FUNCTION_BLOCK EnableCheck (* Template for an empty basic function block *)
  (* Standard: 61499-2 *)
  (* Version 1.0, 2018-06-08, Duc Do Tran, OFFIS e.V. *)
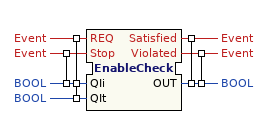
  EVENT_INPUT
    REQ WITH QIi, QIt;
    Stop WITH QIi;
  END_EVENT
  EVENT_OUTPUT
    Satisfied WITH OUT;
    Violated WITH OUT;
  END_EVENT
  VAR_INPUT
    QIi : BOOL := 1; (* QIt *)
    QIt : BOOL;
  END_VAR
  VAR_OUTPUT
    OUT : BOOL;
  END_VAR
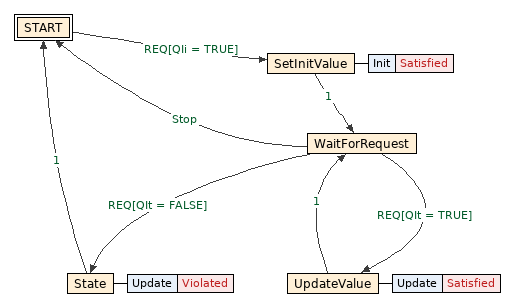
  EC_STATES
    START; (* Initial State *)
    SetInitValue : Init -> Satisfied;
    UpdateValue : Update -> Satisfied;
    WaitForRequest;
    State : Update -> Violated;
  END_STATES
  EC_TRANSITIONS
    START TO SetInitValue := REQ[QIi = TRUE];
    SetInitValue TO WaitForRequest := 1;
    WaitForRequest TO UpdateValue := REQ[QIt = TRUE];
    UpdateValue TO WaitForRequest := 1;
    WaitForRequest TO START := Stop;
    WaitForRequest TO State := REQ[QIt = FALSE];
    State TO START := 1;
  END_TRANSITIONS
  ALGORITHM Init IN ST: (* new algorithm *)
OUT := QIi;
  END_ALGORITHM
  ALGORITHM Update IN ST: (* new algorithm *)
OUT := QIt;
  END_ALGORITHM
END_FUNCTION_BLOCK
